Staubli VAL3: onEnterEvent.pgx

program onEnterEvent(bool& x_bSave[])
  local string l_sItem
  local num l_nValue
  local num l_nMin
  local num l_nMax
  local num l_nValue1
begin
  // look if the bButton is enable
  call axis:get(l_sItem,nIndex)

  call axis:getVelocity(l_sItem,l_nValue)
  if l_sItem!=""
    // change the value
    l_nMin=0.99
    l_nMax=600.01
    call use:insertDialog(l_sItem+"   ",l_nValue,l_nMin,l_nMax)
    call axis:setVelocity(l_nValue,nIndex)
    x_bSave=true
  endIf
  libSave(axis:libPath())
  //
  // NB sEvent is the selected
  // element in the LIST
  //
end
